{attribute 'qualified_only'}
{attribute 'strict'}
TYPE SeqState :
(
	TO_INIT,
	Ready,
	Fill_A,
	Fill_B,
	Heating,
	ToUnload,
	Drain_1,
	Drain_2
	);
END_TYPE

(* stored: Version 1.1.0.1, ProductVersion 3.1.4024.2
   EnumerationTextList SeqState: Id {bb733441-c6d5-49ec-aca8-d1c160e7cfc7} *)
